VAR_GLOBAL CONSTANT // CONSTANTS
    a: DINT := 4;
    b: DINT := 2;
    c: LREAL := 3.0;
    d: DINT := 1;
    holds: BOOL := TRUE;
    danger: Color := red;
    x: DINT := -1;
END_VAR

(* stored: ProductVersion 3.1.0.18, Version 1.1.0.1 *)
